// TIA Portal V17 export
// export: Created 2022-07-20T06:59:49.4418834Z, ExportSetting WithDefaults, DisplayName Totally Integrated Automation Portal, DisplayVersion V17, DisplayName TIA Portal Openness, DisplayVersion V17, DisplayName TIA Portal Version Control Interface, DisplayVersion V17, DisplayName SINAMICS Startdrive Advanced, DisplayVersion V17, DisplayName SINAMICS Startdrive G130, G150, S120, S150, SINAMICS MV, S210, DisplayVersion V17, DisplayName SINAMICS Startdrive G110M, G120, G120C, G120D, G120P, G115D, DisplayVersion V17, DisplayName STEP 7 Professional, DisplayVersion V17, DisplayName STEP 7 Safety, DisplayVersion V17, DisplayName WinCC Advanced, DisplayVersion V17
FUNCTION "FC10020_Linearization" : Void   // FC10020, LAD
{ S7_Optimized_Access := 'TRUE' }
VERSION : 0.1
// stored: AutoNumber false, IsIECCheckEnabled false, SetENOAutomatically false, UDAEnableTagReadback false
   VAR_INPUT
      X1 : Real;
      Y1 : Real;
      X2 : Real;
      Y2 : Real;
      X : Real;
   END_VAR
   VAR_OUTPUT
      Y : Real;
   END_VAR
BEGIN

REGION Network 1 (SCL): Linearization
   IF #X2 - #X1 <> 0 THEN
       #Y := (((#Y2 - #Y1) / (#X2 - #X1)) * #X) + (((#X2 * #Y1) - (#X1 * #Y2)) / (#X2 - #X1));
   ELSE
       #Y := 0;
   END_IF;
END_REGION
END_FUNCTION
